RoboDK station: DynamicTarget.rdk

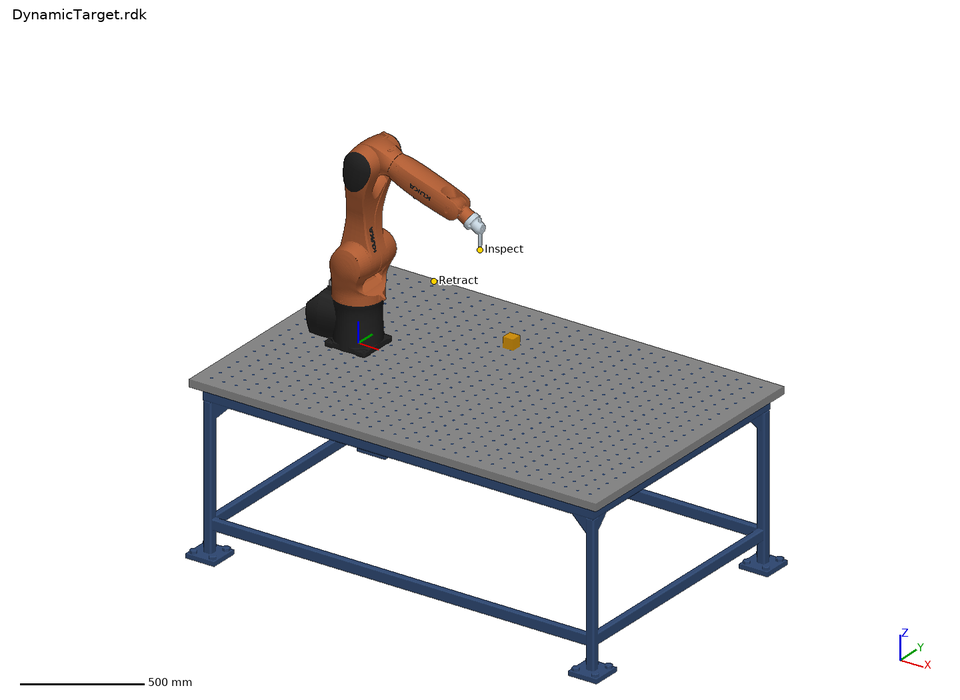
[picture v0: the station drawn from its stored meshes, robots at their saved joint values, targets as dots, program paths as lines]
Station DynamicTarget (saved by RoboDK 5.5.2). Poses are relative to the parent item; angles as X-Y-Z fixed-axis rotations.
  - frame Base at (-207.87, 0, -62.35) mm
    - robot Robot (model KUKA KR 6 R900 sixx): 6 axes, payload 6 kg, reach 901 mm, repeatability 0.03 mm, weight 52 kg
        modified DH rows (alpha deg, a mm, theta deg, d mm): 0, 0, 0, 400; -90, 25, 0, 0; 0, 455, -90, 0; -90, 35, 0, 420; 90, 0, 0, 0; -90, 0, 180, 80
        joint limits [-170, -190, -120, -185, -120, -350] to [170, 45, 156, 185, 120, 350]; home [0, -90, 90, 0, 0, 0]; saved at [-0.299, -84.178, 103.493, 181.395, -10.689, -181.52]
      - tool Pencil, TCP at (82.2, 0, 101.78) mm, rotated rx 0 ry 60 rz 0 deg, size 74.9 x 125 x 107.3 mm
    - target Retract (Cartesian target) at (370.47, 2.5, 379.03) mm, rotated rx 180 ry 0 rz -180 deg; joints [-0.563, -97.056, 149.262, 178.71, 22.21, -179.087] of Robot
    - target Inspect (Cartesian target) at (595.41, 2.5, 584.69) mm, rotated rx 180 ry 0 rz -180 deg; joints [-0.299, -84.178, 103.493, 181.395, -10.689, -181.52] of Robot
    - object Cube at (500, 300, 0) mm, size 50 x 50 x 50 mm, geometry from Cube-50mm.sld
    - object Table at (0, 0, 0) mm, size 2020 x 1340 x 800 mm, geometry from Table-2000x1200x800mm.sld
  - Python program dynamicTarget (listed below)

--- Python program dynamicTarget ---
from robodk.robolink import *      # RoboDK's API
from robodk.robomath import *      # Math toolbox for robots
from graphic_interface import interface

RL = Robolink()

robot = RL.Item('Robot')
base = RL.Item('Base')
inspect = RL.Item('Inspect')
retract = RL.Item('Retract')

target = RL.AddTarget('Cube', base)
center = interface()
RL.ShowMessage('Centers: ' + str(center))
target.setPose(Offset(eye(), 600, -100, 0, -180, 0, 180))

robot.MoveJ(inspect)
robot.MoveJ(target)
robot.MoveJ(retract)
